TYPE ST_Auto_UpperFeedInConveyorStatus EXTENDS ST_StatusBasic :
STRUCT
END_STRUCT
END_TYPE

(* stored: Version 1.1.0.1, ProductVersion 3.1.4024.13
   DUT ST_Auto_UpperFeedInConveyorStatus: Id {fbc7f4f2-9723-4728-8f08-298d10cd7d64} *)
